PROGRAM Horizontal_Sample
VAR
END_VAR

astAxes[AXIS_HORIZONTAL_SAMPLE].stControl.bEnable := TRUE;
astAxes[AXIS_HORIZONTAL_SAMPLE].stInputs.bLimitBwd := astAxes[AXIS_HORIZONTAL_TRANSLATION].stInputs.bLimitBwd;
astAxes[AXIS_HORIZONTAL_SAMPLE].stInputs.bLimitFwd := astAxes[AXIS_HORIZONTAL_TRANSLATION].stInputs.bLimitFwd;

astAxes[AXIS_HORIZONTAL_SAMPLE].stDescription.sAxisName := 'SAMPLE_HORIZ';

END_PROGRAM

(* stored: Version 1.1.0.1, ProductVersion 3.1.4024.12
   POU Horizontal_Sample: Id {33e2f27d-2a6a-4757-a88a-96a036297ac6}, SpecialFunc None *)
